// TIA Portal V19 export
DATA_BLOCK "Flow Count"   // DB7
{ S7_Optimized_Access := 'TRUE' }
// stored: AutoNumber false, MemoryReserve 0
   VAR RETAIN
      Prod_Vol_Count : Real := 0.0;   // Product Volume to Hamba2/Gasti
   END_VAR
BEGIN
END_DATA_BLOCK
